// PLC-owned exchange boundary for the complete discrete assembly station.
// Python supplies one coherent plant-input frame; this cyclic owner alone runs
// the controller and publishes its six output coils.
FUNCTION_BLOCK FB_SimulationBridge
VAR_INPUT
    recoverOnOnlineChange : BOOL := TRUE;
END_VAR

VAR_OUTPUT
    outClampAdvance, outClampRetract : BOOL;
    outPressAdvance, outPressRetract : BOOL;
    outEjectorAdvance, outEjectorRetract : BOOL;
END_VAR

VAR
    continuity : TcForge.FB_ExecutionContinuity;
    machine : FB_AssemblyStation;
    stationInputs : ST_AssemblyInputs;
    mutex : BOOL;
    boot, cycle, session, submitted, applied, lastAck : ULINT;
    pending, hasFrame, freshPrevious, newClaim : BOOL;
    pendingClampAdvanced, pendingClampRetracted : BOOL;
    pendingPressAdvanced, pendingPressRetracted : BOOL;
    pendingEjectorAdvanced, pendingEjectorRetracted : BOOL;
    pendingPartPresent, pendingDischargeClear : BOOL;
    pendingShutdown, pendingQuality : BOOL;
    pendingPressureRaw, pendingHeightRaw : INT;
    pendingCommand : UINT;
    command : E_ReferenceCommand;
    quality : TcForge.E_IO_Quality;
    watchdog : TON;
    owner : DINT;
    ownershipConflict : BOOL;
END_VAR

// 1. Serialize RPC exchange state with the owning PLC task.
IF NOT Tc2_System.TestAndSet(mutex) THEN
    RETURN;
END_IF;
IF owner = 0 THEN
    owner := Tc2_System.GETCURTASKINDEXEX();
    IF owner <= 0 THEN
        owner := 0;
        mutex := FALSE;
        RETURN;
    END_IF;
    boot := Tc2_System.F_GetSystemTime();
END_IF;
IF Tc2_System.GETCURTASKINDEXEX() <> owner THEN
    ownershipConflict := TRUE;
    session := 0;
    pending := FALSE;
    hasFrame := FALSE;
    outClampAdvance := FALSE;
    outClampRetract := FALSE;
    outPressAdvance := FALSE;
    outPressRetract := FALSE;
    outEjectorAdvance := FALSE;
    outEjectorRetract := FALSE;
    mutex := FALSE;
    RETURN;
END_IF;

// 2. Any execution gap rotates the epoch and discards unconsumed input.
continuity(
    taskIndex := owner,
    cycleCounter := TwinCAT_SystemInfoVarList._TaskInfo[owner].CycleCount,
    onlineChangeCounter := TwinCAT_SystemInfoVarList._AppInfo.OnlineChangeCnt,
    recoverOnOnlineChange := recoverOnOnlineChange
);
IF continuity.interrupted THEN
    boot := Tc2_System.F_GetSystemTime();
    session := 0;
    pending := FALSE;
    hasFrame := FALSE;
    freshPrevious := FALSE;
    newClaim := FALSE;
    submitted := 0;
    applied := 0;
    lastAck := 0;
    pendingCommand := 0;
    watchdog(IN := FALSE, PT := T#250MS);
END_IF;

// 3. Expire stale writers independently of the Python process.
watchdog(IN := session <> 0 AND NOT freshPrevious, PT := T#250MS);
freshPrevious := FALSE;
IF newClaim THEN
    watchdog(IN := FALSE, PT := T#250MS);
    newClaim := FALSE;
END_IF;
IF watchdog.Q OR ownershipConflict THEN
    session := 0;
    pending := FALSE;
    hasFrame := FALSE;
END_IF;

// 4. Apply an admitted frame atomically at the scan boundary.
command := E_ReferenceCommand.None;
IF pending AND session <> 0 THEN
    stationInputs.clamp.advanced := pendingClampAdvanced;
    stationInputs.clamp.retracted := pendingClampRetracted;
    stationInputs.press.advanced := pendingPressAdvanced;
    stationInputs.press.retracted := pendingPressRetracted;
    stationInputs.ejector.advanced := pendingEjectorAdvanced;
    stationInputs.ejector.retracted := pendingEjectorRetracted;
    stationInputs.partPresent := pendingPartPresent;
    stationInputs.dischargeClear := pendingDischargeClear;
    stationInputs.pressureRaw := pendingPressureRaw;
    stationInputs.heightRaw := pendingHeightRaw;
    stationInputs.shutdownConfirmed := pendingShutdown;
    CASE pendingCommand OF
        1: command := E_ReferenceCommand.Home;
        2: command := E_ReferenceCommand.Start;
        3: command := E_ReferenceCommand.Stop;
        4: command := E_ReferenceCommand.Abort;
        5: command := E_ReferenceCommand.Reset;
    END_CASE;
    applied := submitted;
    pending := FALSE;
    hasFrame := TRUE;
    freshPrevious := TRUE;
END_IF;

IF hasFrame AND session <> 0 AND pendingQuality AND NOT ownershipConflict THEN
    quality := TcForge.E_IO_Quality.GOOD;
ELSE
    quality := TcForge.E_IO_Quality.BAD;
END_IF;
stationInputs.inputQuality := quality;
stationInputs.outputQuality := quality;
stationInputs.shutdownQuality := quality;

// 5. The production-style controller runs every available PLC scan.
machine(
    inputs := stationInputs,
    command := command,
    recoverOnOnlineChange := recoverOnOnlineChange
);
outClampAdvance := machine.outputs.clamp.advance AND quality = TcForge.E_IO_Quality.GOOD;
outClampRetract := machine.outputs.clamp.retract AND quality = TcForge.E_IO_Quality.GOOD;
outPressAdvance := machine.outputs.press.advance AND quality = TcForge.E_IO_Quality.GOOD;
outPressRetract := machine.outputs.press.retract AND quality = TcForge.E_IO_Quality.GOOD;
outEjectorAdvance := machine.outputs.ejector.advance AND quality = TcForge.E_IO_Quality.GOOD;
outEjectorRetract := machine.outputs.ejector.retract AND quality = TcForge.E_IO_Quality.GOOD;
cycle := cycle + 1;
mutex := FALSE;

{attribute 'TcRpcEnable' := '1'}
METHOD PUBLIC Identity : STRING(80)
Identity := 'TcForge.DiscreteAssembly/2';
END_METHOD

{attribute 'TcRpcEnable' := '1'}
METHOD PUBLIC Claim : DINT
VAR_INPUT
    client : ULINT;
    expectedBoot : ULINT;
END_VAR
Claim := 30;
IF client = 0 THEN RETURN; END_IF;
Claim := 22;
IF NOT Tc2_System.TestAndSet(mutex) THEN RETURN; END_IF;
IF boot = 0 OR owner = 0 THEN
    Claim := 12;
ELSIF ownershipConflict THEN
    Claim := 13;
ELSIF expectedBoot <> boot THEN
    Claim := 34;
ELSIF session <> 0 THEN
    IF client = session THEN Claim := 0; ELSE Claim := 11; END_IF;
ELSE
    session := client;
    submitted := 0;
    applied := 0;
    lastAck := 0;
    pending := FALSE;
    hasFrame := FALSE;
    newClaim := TRUE;
    Claim := 0;
END_IF;
mutex := FALSE;
END_METHOD

{attribute 'TcRpcEnable' := '1'}
METHOD PUBLIC Exchange : DINT
VAR_INPUT
    client, expectedBoot, frame, outputFrame : ULINT;
    clampAdvanced, clampRetracted : BOOL;
    pressAdvanced, pressRetracted : BOOL;
    ejectorAdvanced, ejectorRetracted : BOOL;
    partPresent, dischargeClear : BOOL;
    pressureRaw, heightRaw : INT;
    shutdownConfirmed, qualityGood : BOOL;
    requestedCommand : UINT;
END_VAR
Exchange := 30;
IF client = 0 OR frame = 0 OR requestedCommand > 5 THEN RETURN; END_IF;
Exchange := 22;
IF NOT Tc2_System.TestAndSet(mutex) THEN RETURN; END_IF;
IF expectedBoot <> boot THEN
    Exchange := 34;
ELSIF session = 0 OR watchdog.Q THEN
    Exchange := 12;
ELSIF client <> session THEN
    Exchange := 11;
ELSIF frame <= submitted THEN
    Exchange := 35;
ELSIF frame <> submitted + 1 OR outputFrame <= lastAck OR outputFrame > cycle THEN
    Exchange := 30;
ELSIF NOT pending THEN
    pendingClampAdvanced := clampAdvanced;
    pendingClampRetracted := clampRetracted;
    pendingPressAdvanced := pressAdvanced;
    pendingPressRetracted := pressRetracted;
    pendingEjectorAdvanced := ejectorAdvanced;
    pendingEjectorRetracted := ejectorRetracted;
    pendingPartPresent := partPresent;
    pendingDischargeClear := dischargeClear;
    pendingPressureRaw := pressureRaw;
    pendingHeightRaw := heightRaw;
    pendingShutdown := shutdownConfirmed;
    pendingQuality := qualityGood;
    pendingCommand := requestedCommand;
    submitted := frame;
    lastAck := outputFrame;
    pending := TRUE;
    Exchange := 1;
END_IF;
mutex := FALSE;
END_METHOD

{attribute 'TcRpcEnable' := '1'}
METHOD PUBLIC Release : DINT
VAR_INPUT
    client, expectedBoot : ULINT;
END_VAR
Release := 22;
IF NOT Tc2_System.TestAndSet(mutex) THEN RETURN; END_IF;
IF expectedBoot <> boot THEN
    Release := 34;
ELSIF session = 0 OR client <> session THEN
    Release := 11;
ELSE
    session := 0;
    hasFrame := FALSE;
    pending := FALSE;
    Release := 0;
END_IF;
mutex := FALSE;
END_METHOD

{attribute 'TcRpcEnable' := '1'}
METHOD PUBLIC Snapshot : STRING(255)
Snapshot := '22';
IF NOT Tc2_System.TestAndSet(mutex) THEN RETURN; END_IF;
Snapshot := '0';
Snapshot := CONCAT(Snapshot, CONCAT(',', ULINT_TO_STRING(boot)));
Snapshot := CONCAT(Snapshot, CONCAT(',', ULINT_TO_STRING(cycle)));
Snapshot := CONCAT(Snapshot, CONCAT(',', ULINT_TO_STRING(applied)));
Snapshot := CONCAT(Snapshot, CONCAT(',', DINT_TO_STRING(BOOL_TO_UINT(outClampAdvance))));
Snapshot := CONCAT(Snapshot, CONCAT(',', DINT_TO_STRING(BOOL_TO_UINT(outClampRetract))));
Snapshot := CONCAT(Snapshot, CONCAT(',', DINT_TO_STRING(BOOL_TO_UINT(outPressAdvance))));
Snapshot := CONCAT(Snapshot, CONCAT(',', DINT_TO_STRING(BOOL_TO_UINT(outPressRetract))));
Snapshot := CONCAT(Snapshot, CONCAT(',', DINT_TO_STRING(BOOL_TO_UINT(outEjectorAdvance))));
Snapshot := CONCAT(Snapshot, CONCAT(',', DINT_TO_STRING(BOOL_TO_UINT(outEjectorRetract))));
Snapshot := CONCAT(Snapshot, CONCAT(',', DINT_TO_STRING(machine.sequence.State)));
Snapshot := CONCAT(Snapshot, CONCAT(',', DINT_TO_STRING(BOOL_TO_UINT(machine.sequence.Faulted))));
Snapshot := CONCAT(Snapshot, CONCAT(',', DINT_TO_STRING(BOOL_TO_UINT(machine.outputsInhibited))));
Snapshot := CONCAT(Snapshot, CONCAT(',', DINT_TO_STRING(machine.lastResponse)));
Snapshot := CONCAT(Snapshot, CONCAT(',', ULINT_TO_STRING(session)));
Snapshot := CONCAT(Snapshot, CONCAT(',', DINT_TO_STRING(owner)));
Snapshot := CONCAT(Snapshot, CONCAT(',', DINT_TO_STRING(BOOL_TO_UINT(quality = TcForge.E_IO_Quality.GOOD AND NOT watchdog.Q))));
Snapshot := CONCAT(Snapshot, CONCAT(',', DINT_TO_STRING(machine.sequence.Step.Current)));
mutex := FALSE;
END_METHOD

END_FUNCTION_BLOCK

(* stored: Version 1.1.0.1
   POU FB_SimulationBridge: Id {cda7da18-db35-40a0-8f86-d99f1451774a}
   Method Identity: Id {ab63e9a4-1390-4f2e-ae93-85a29b4a1195}
   Method Claim: Id {7aa0e04b-4453-4956-9032-c6c93b2f5913}
   Method Exchange: Id {4e3fa12d-8736-422b-a284-c8d3e4777168}
   Method Release: Id {bc1d824f-c731-4236-a795-9dd4b0530cb9}
   Method Snapshot: Id {88648abe-099f-4e5f-83a2-895a0c4b98e0} *)
